# EPICS autosave request: 3-4/GalilSup/Db/galil_digital_in_bit.req
$(P)$(R)_STATUS.DESC
